{attribute 'qualified_only'}
TYPE E_OpMod_Step2 :
(
	Invalid			:= 0,
	
	eOff			:= 1,
	eStep1			:= 2,
	eStep2			:= 3
	
) UDINT;
END_TYPE

(* stored: Version 1.1.0.1, ProductVersion 3.1.4024.5
   DUT E_OpMod_Step2: Id {580cf63d-08ed-4c9c-88b2-945ac669afc5} *)
